FUNCTION_BLOCK PRESS (* Modell of a simple mechanical press *)
  (* Standard: 61499-2 *)
  (* Version 0.2, 2003-12-05, JHC, Rockwell Automation, Renamed from NEWCOMPFB. *)
  (* Version 0.1, 2002-01-08, JHC, Rockwell Automation, Added DLY FB as example. *)
  (* Version 0.0, 2000-05-27, JHC, Rockwell Automation *)
  (* Compiler header: package fb.rt.mach; import fb.rt.mva.*; *)
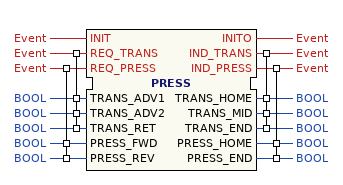
  EVENT_INPUT
    INIT; (* Initialization Request *)
    REQ_TRANS WITH TRANS_ADV1, TRANS_ADV2, TRANS_RET; (* Request command for transport unit *)
    REQ_PRESS WITH PRESS_FWD, PRESS_REV; (* Request command for press unit *)
  END_EVENT
  EVENT_OUTPUT
    INITO; (* Initialization Confirm *)
    IND_TRANS WITH TRANS_HOME, TRANS_MID, TRANS_END; (* Sensors of transport unit have changed *)
    IND_PRESS WITH PRESS_HOME, PRESS_END; (* Sensors of press unit have changed *)
  END_EVENT
  VAR_INPUT
    TRANS_ADV1 : BOOL; (* Advance transport unit to position 1 (middle position), must be true until position MID is reachted *)
    TRANS_ADV2 : BOOL; (* Advance transport unit to position 2 (end position), must be true until position END is reachted *)
    TRANS_RET : BOOL; (* Advance transport unit back to home position, must be true until position HOME is reachted *)
    PRESS_FWD : BOOL; (* Advance press forward, must be true until position END is reachted *)
    PRESS_REV : BOOL; (* Advance press backward, must be true until position HOME is reachted *)
  END_VAR
  VAR_OUTPUT
    TRANS_HOME : BOOL; (* Transport is in HOME postion *)
    TRANS_MID : BOOL; (* Transport is in MID postion *)
    TRANS_END : BOOL; (* Transport is in END postion *)
    PRESS_HOME : BOOL; (* Press is in HOME postion *)
    PRESS_END : BOOL; (* Press is in END postion *)
  END_VAR
  FBS
    CLCK : E_CYCLE(DT := t#250ms);
    SP1 : XSPACE(LBLS := ["","",PART2,PART1], DIMS := [3,3], DIA := 25);
    SP2 : XSPACE(LBLS := [PressFit,"","",Transport], DIMS := [3,3], DIA := 25);
    PRESS_VIEW : MECH_VIEW(LEN := 3, DIA := 25, DIR := 1, BKGD := COLOR#gray);
    TRANSPORT_VIEW : MECH_VIEW(LEN := 7, DIA := 25, DIR := 0);
    TRANSPORT_MODEL : DSCYL_MDL(VF1 := 10, VF2 := 10, VR := 10, ETA := 0.5);
    TRANSPORT_LDU : E_LDU(S0 := VSTYLE#EMPTY);
    UNLOAD_TRANS : E_R_TRIG;
    LD_TRANS : E_R_TRIG;
    PRESS_MODEL : MECH2_MDL(VF := 10, VR := 10);
    PRESS_LDU : E_LDU(S0 := VSTYLE#EMPTY, W1 := [255,0,255], S1 := VSTYLE#RING);
    UNLOAD_PRESS : E_R_TRIG;
    LD_PRESS : E_R_TRIG;
    TRANSPORT_PRESSED : E_LDU(S1 := VSTYLE#PEG, S0 := VSTYLE#PEGRING, W1 := [255,0,255]);
  END_FBS
  EVENT_CONNECTIONS
    SP1.INITO TO PRESS_VIEW.INIT;
    PRESS_VIEW.INITO TO SP2.INIT;
    SP2.INITO TO TRANSPORT_VIEW.INIT;
    CLCK.EO TO TRANSPORT_MODEL.CLK;
    TRANSPORT_MODEL.INDP TO TRANSPORT_VIEW.REQ;
    TRANSPORT_MODEL.INDS TO UNLOAD_TRANS.EI;
    UNLOAD_TRANS.EO TO TRANSPORT_LDU.UNLD;
    TRANSPORT_MODEL.INDS TO LD_TRANS.EI;
    CLCK.EO TO PRESS_MODEL.CLK;
    PRESS_MODEL.INDP TO PRESS_VIEW.REQ;
    PRESS_MODEL.INDS TO UNLOAD_PRESS.EI;
    UNLOAD_PRESS.EO TO PRESS_LDU.UNLD;
    PRESS_MODEL.INDS TO LD_PRESS.EI;
    LD_PRESS.EO TO PRESS_LDU.LD1;
    PRESS_LDU.LD TO PRESS_VIEW.REQ;
    TRANSPORT_LDU.LD TO TRANSPORT_VIEW.REQ;
    LD_TRANS.EO TO TRANSPORT_PRESSED.LD1;
    TRANSPORT_PRESSED.LD TO TRANSPORT_LDU.LD1;
    UNLOAD_PRESS.EO TO TRANSPORT_PRESSED.UNLD;
    INIT TO SP1.INIT;
    PRESS_MODEL.INDS TO IND_PRESS;
    TRANSPORT_VIEW.INITO TO TRANSPORT_PRESSED.LD1;
    TRANSPORT_VIEW.INITO TO PRESS_LDU.LD1;
    TRANSPORT_VIEW.INITO TO CLCK.START;
    TRANSPORT_VIEW.INITO TO INITO;
    TRANSPORT_MODEL.INDS TO IND_TRANS;
  END_CONNECTIONS
  DATA_CONNECTIONS
    TRANSPORT_VIEW.FAULT TO TRANSPORT_MODEL.FAULT;
    TRANSPORT_MODEL.POS TO TRANSPORT_VIEW.POS;
    TRANSPORT_LDU.STYLE TO TRANSPORT_VIEW.STYLE;
    TRANSPORT_LDU.WKPC TO TRANSPORT_VIEW.WKPC;
    TRANSPORT_MODEL.END TO UNLOAD_TRANS.QI;
    TRANSPORT_MODEL.HOME TO LD_TRANS.QI;
    PRESS_MODEL.POS TO PRESS_VIEW.POS;
    PRESS_VIEW.FAULT TO PRESS_MODEL.FAULT;
    PRESS_LDU.STYLE TO PRESS_VIEW.STYLE;
    PRESS_LDU.WKPC TO PRESS_VIEW.WKPC;
    PRESS_MODEL.END TO UNLOAD_PRESS.QI;
    PRESS_MODEL.HOME TO LD_PRESS.QI;
    TRANSPORT_PRESSED.STYLE TO TRANSPORT_LDU.S1;
    TRANSPORT_PRESSED.WKPC TO TRANSPORT_LDU.W1;
    PRESS_MODEL.HOME TO PRESS_HOME;
    PRESS_MODEL.END TO PRESS_END;
    PRESS_FWD TO PRESS_MODEL.FWD;
    PRESS_REV TO PRESS_MODEL.REV;
    TRANS_ADV1 TO TRANSPORT_MODEL.ADV1;
    TRANS_ADV2 TO TRANSPORT_MODEL.ADV2;
    TRANS_RET TO TRANSPORT_MODEL.RET;
    TRANSPORT_MODEL.HOME TO TRANS_HOME;
    TRANSPORT_MODEL.MID TO TRANS_MID;
    TRANSPORT_MODEL.END TO TRANS_END;
  END_CONNECTIONS
END_FUNCTION_BLOCK
